ABB RobotStudio station: LAB1.rspag

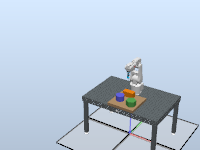
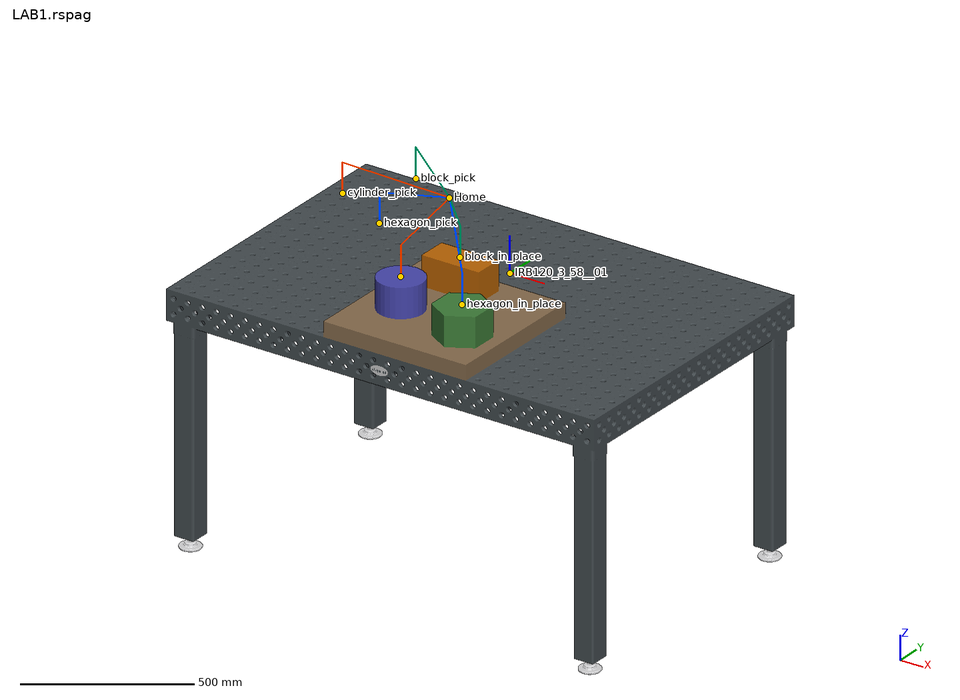
[picture v1: parts stored in the station drawn from their meshes, with robot base, taught points and paths (robot models come from the ABB library and are not in the file)]
--- station ---
Station Solution_1_Tutorial (saved by RobotStudio 21.4.9700.0)
Controller Controller1, task T_ROB1: task frame (RAPID world) sits at (0, 150, 830) mm, rotated rx 0 ry 0 rz -90 deg in the station
Controller Controller1
  mechanical unit ROB_1: IRB120_3_58__01, 6 joints, base frame (0, 0, 0) mm
Layout (positions relative to the parent item):
  - table [part] at (-200, -500, 830) mm, size 500 x 500 x 50 mm
  - Block [part] at (-200, -500, 830) mm, size 200 x 100 x 150 mm
  - Cylindric [part] at (-200, -500, 830) mm, size 149.5 x 149.7 x 150 mm
  - Hexagon [part] at (-200, -500, 830) mm, size 155.5 x 179.5 x 150 mm
  - siegmund_1500_1000 [part], size 1500 x 1010.3 x 830 mm
  - Block1 [part] at (-200, -500, 830) mm, size 200 x 100 x 150 mm
  - Cylinder1 [part] at (-200, -500, 830) mm, size 149.5 x 149.7 x 150 mm
  - Hexagon1 [part] at (-200, -500, 830) mm, size 155.5 x 179.5 x 150 mm
  - IRB120_3_58__01 [mechanism, from Robots\IRB120_3_58_G_01.rslib] at (0, 150, 830) mm, rotated rx 0 ry 0 rz -90 deg; joint values [0, 0, 0, 0, 1.5708, 0] (rad or m)
  - smc_gripper [mechanism, from Lab1\smc_gripper.rslib] at (0, -152, 1388) mm, rotated rx 180 ry 0 rz 90 deg
  - Positioner_2 [smart component, from Components\Positioner.rslib]
      properties: Object=Hexagon; Position=[-0.7 -0.2 0.83]; Orientation=[0 0 0]; Reference=Global; ReferenceObject=(none)
  - Positioner_3 [smart component, from Components\Positioner.rslib]
      properties: Object=Block; Position=[-0.6 -0.15 0.83]; Orientation=[0 0 0]; Reference=Global; ReferenceObject=(none)
  - Positioner_4 [smart component, from Components\Positioner.rslib]
      properties: Object=Cylindric; Position=[-0.65 -0.15 0.83]; Orientation=[0 0 0]; Reference=Global; ReferenceObject=(none)
  - Attacher [smart component, from Components\Attacher.rslib]
      properties: Parent=smc_gripper; Flange=0; Child=Hexagon; Mount=false; Offset=[0 0 0]; Orientation=[0 0 0]
  - Detacher [smart component, from Components\Detacher.rslib]
      properties: Child=Hexagon; KeepPosition=true
  - Attacher_2 [smart component, from Components\Attacher.rslib]
      properties: Parent=smc_gripper; Flange=0; Child=Cylindric; Mount=false; Offset=[0 0 0]; Orientation=[0 0 0]
  - Detacher_2 [smart component, from Components\Detacher.rslib]
      properties: Child=Cylindric; KeepPosition=true
  - Attacher_3 [smart component, from Components\Attacher.rslib]
      properties: Parent=smc_gripper; Flange=0; Child=Block; Mount=false; Offset=[0 0 0]; Orientation=[0 0 0]
  - Detacher_3 [smart component, from Components\Detacher.rslib]
      properties: Child=Block; KeepPosition=true
Attachment: smc_gripper is attached to IRB120_3_58__01 / Link6
Station signals: DI hexagon, DI cylinder, DI block
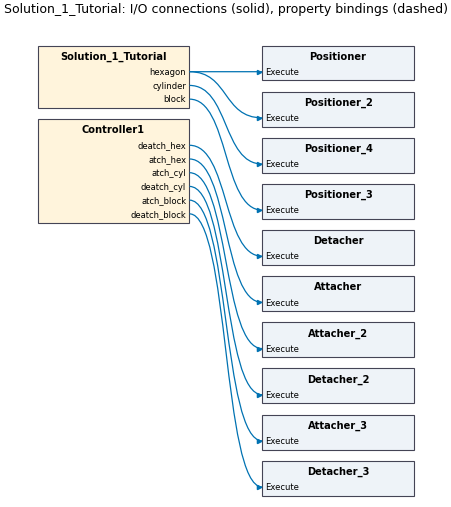
Station logic (signal -> signal, property => property):
  Solution_1_Tutorial.hexagon -> Positioner.Execute
  Solution_1_Tutorial.hexagon -> Positioner_2.Execute
  Solution_1_Tutorial.cylinder -> Positioner_4.Execute
  Solution_1_Tutorial.block -> Positioner_3.Execute
  Controller1.deatch_hex -> Detacher.Execute
  Controller1.atch_hex -> Attacher.Execute
  Controller1.atch_cyl -> Attacher_2.Execute
  Controller1.deatch_cyl -> Detacher_2.Execute
  Controller1.atch_block -> Attacher_3.Execute
  Controller1.deatch_block -> Detacher_3.Execute
Targets, tools, work objects and paths stored in the station and not in the controller backup, written as RAPID:
! task (no controller)
MODULE Module1
  CONST robtarget Target_10:=[[-317.298,-50,980],[1,0,0,0],[0,0,0,0],[9E+09,9E+09,9E+09,9E+09,9E+09,9E+09]];
  CONST robtarget Target_20:=[[-517.298,50,980],[1,0,0,0],[0,0,0,0],[9E+09,9E+09,9E+09,9E+09,9E+09,9E+09]];
  CONST robtarget Target_30:=[[-400,250,980],[1,0,0,0],[0,0,0,0],[9E+09,9E+09,9E+09,9E+09,9E+09,9E+09]];
  CONST robtarget Target_40:=[[0,-100,980],[1,0,0,0],[0,0,0,0],[9E+09,9E+09,9E+09,9E+09,9E+09,9E+09]];
  CONST robtarget Target_50:=[[-67.298,-300,980],[1,0,0,0],[0,0,0,0],[9E+09,9E+09,9E+09,9E+09,9E+09,9E+09]];
  CONST robtarget Target_60:=[[182.702,-350,980],[1,0,0,0],[0,0,0,0],[9E+09,9E+09,9E+09,9E+09,9E+09,9E+09]];
ENDMODULE


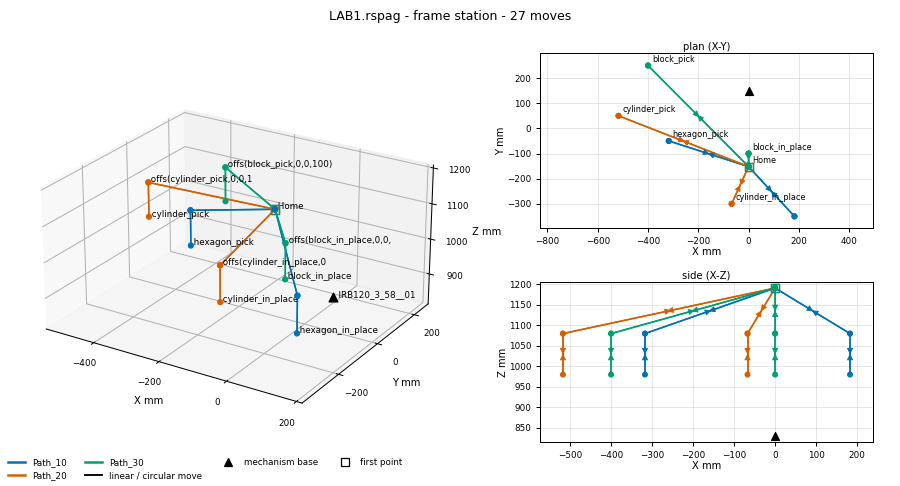
[picture p0: tool path of LAB1.rspag in frame station, 27 of 27 moves have a stored position in this frame; points joined in program order, loops and branches not executed]
--- Backups/Controller1/RAPID/TASK1/PROGMOD/CalibData.mod ---
MODULE CalibData
    PERS tooldata smc_gripper:=[TRUE,[[0,0.004,197.001],[1,0,0,0]],[1,[0.207,-0.496,71.18],[1,0,0,0],0,0,0]];
ENDMODULE

--- Backups/Controller1/RAPID/TASK1/PROGMOD/Module1.mod ---
MODULE Module1
    CONST robtarget hexagon_pick:=[[200,-317.298,150],[0.000022965,0,1,0],[-1,0,-1,0],[9E+09,9E+09,9E+09,9E+09,9E+09,9E+09]];
    CONST robtarget Home:=[[302.01235514,0.004,360.999000284],[0.000022965,0,1,0],[-1,0,-1,0],[9E+09,9E+09,9E+09,9E+09,9E+09,9E+09]];
    CONST robtarget hexagon_in_place:=[[500,182.702,150],[0.000022965,0,1,0],[0,0,0,0],[9E+09,9E+09,9E+09,9E+09,9E+09,9E+09]];
    CONST robtarget block_pick:=[[-100,-400,150],[0.000022965,0,1,0],[0,0,0,0],[9E+09,9E+09,9E+09,9E+09,9E+09,9E+09]];
    CONST robtarget block_in_place:=[[250,0,150],[0.000022965,0,1,0],[-1,0,-1,0],[9E+09,9E+09,9E+09,9E+09,9E+09,9E+09]];
    CONST robtarget cylinder_pick:=[[100,-517.298,150],[0.000022965,0,1,0],[-1,0,-1,0],[9E+09,9E+09,9E+09,9E+09,9E+09,9E+09]];
    CONST robtarget cylinder_in_place:=[[450,-67.298,150],[0.000022965,0,1,0],[-1,0,-1,0],[9E+09,9E+09,9E+09,9E+09,9E+09,9E+09]];


    PROC main()
        Path_10;
        Path_20;
        Path_30;

    ENDPROC
    PROC Path_10()
        MoveL Home,v200,fine,smc_gripper\WObj:=wobj0;
        MoveL offs(hexagon_pick,0,0,100),v200,fine,smc_gripper\WObj:=wobj0;
        MoveL hexagon_pick,v200,fine,smc_gripper\WObj:=wobj0;

        WaitTime 0.1;
        PulseDO atch_hex;
        WaitTime 0.1;

        MoveL offs(hexagon_pick,0,0,100),v200,fine,smc_gripper\WObj:=wobj0;
        MoveL Home,v200,fine,smc_gripper\WObj:=wobj0;

        MoveL offs(hexagon_in_place,0,0,100),v200,fine,smc_gripper\WObj:=wobj0;
        MoveL hexagon_in_place,v200,fine,smc_gripper\WObj:=wobj0;

        WaitTime 0.1;
        PulseDO deatch_hex;
        WaitTime 0.1;
        MoveL offs(hexagon_in_place,0,0,100),v200,fine,smc_gripper\WObj:=wobj0;
        MoveL Home,v200,fine,smc_gripper\WObj:=wobj0;

    ENDPROC
    PROC Path_20()
        MoveL Home,v200,fine,smc_gripper\WObj:=wobj0;
        MoveL offs(cylinder_pick,0,0,100),v200,fine,smc_gripper\WObj:=wobj0;
        MoveL cylinder_pick,v200,fine,smc_gripper\WObj:=wobj0;

        WaitTime 0.1;
        PulseDO atch_cyl;
        WaitTime 0.1;

        MoveL offs(cylinder_pick,0,0,100),v200,fine,smc_gripper\WObj:=wobj0;
        MoveL Home,v200,fine,smc_gripper\WObj:=wobj0;

        MoveL offs(cylinder_in_place,0,0,100),v200,fine,smc_gripper\WObj:=wobj0;
        MoveL cylinder_in_place,v200,fine,smc_gripper\WObj:=wobj0;

        WaitTime 0.1;
        PulseDO deatch_cyl;
        WaitTime 0.1;
        MoveL offs(cylinder_in_place,0,0,100),v200,fine,smc_gripper\WObj:=wobj0;
        MoveL Home,v200,fine,smc_gripper\WObj:=wobj0;
    ENDPROC

    PROC Path_30()
        MoveL Home,v200,fine,smc_gripper\WObj:=wobj0;
        MoveL offs(block_pick,0,0,100),v200,fine,smc_gripper\WObj:=wobj0;
        MoveL block_pick,v200,fine,smc_gripper\WObj:=wobj0;

        WaitTime 0.1;
        PulseDO atch_block;
        WaitTime 0.1;

        MoveL offs(block_pick,0,0,100),v200,fine,smc_gripper\WObj:=wobj0;
        MoveL Home,v200,fine,smc_gripper\WObj:=wobj0;

        MoveL offs(block_in_place,0,0,100),v200,fine,smc_gripper\WObj:=wobj0;
        MoveL block_in_place,v200,fine,smc_gripper\WObj:=wobj0;

        WaitTime 0.1;
        PulseDO deatch_block;
        WaitTime 0.1;
        MoveL offs(block_in_place,0,0,100),v200,fine,smc_gripper\WObj:=wobj0;
        MoveL Home,v200,fine,smc_gripper\WObj:=wobj0;
    ENDPROC
ENDMODULE

--- Backups/Controller1/SYSPAR/EIO.cfg ---
EIO:CFG_1.0:6:1::
#
EIO_SIGNAL:

      -Name "hexagon" -SignalType "DO"

      -Name "deatch_hex" -SignalType "DO"

      -Name "deatch_block" -SignalType "DO"

      -Name "deatch_cyl" -SignalType "DO"

      -Name "atch_hex" -SignalType "DO"

      -Name "atch_block" -SignalType "DO"

      -Name "atch_cyl" -SignalType "DO"
